TYPE T_Ctrl_SIf_MOD_In :
STRUCT
	// Inputs from global module for general supervision 
	// Emergency circuit ok
	bolEmergencyOffOk: T_Ctrl_IoBool;
	// No general error active, will be set to FALSE if there is an global error like e.g. over temperature in cabinet. 
	bolNoGeneralError: T_Ctrl_IoBool;
END_STRUCT
END_TYPE

(* stored: Version 1.1.0.1, ProductVersion 3.1.0.19
   DUT T_Ctrl_SIf_MOD_In: Id {c5b15054-e67d-4931-8724-08ea80cbc6e4} *)
